FUNCTION fcHMIBit : BOOL
VAR_INPUT
	bInToggle:BOOL;
	bInLatch:BOOL;
END_VAR
VAR_IN_OUT
	bHMI:BOOL;
	bPLC:BOOL;
END_VAR

(*set bPLC when bHMI set*)

IF bHMI AND NOT(bPLC) THEN
	bPLC:=1;
	bHMI:=0;
END_IF

END_FUNCTION

(* stored: Version 1.1.0.1, ProductVersion 3.1.4024.11
   POU fcHMIBit: Id {aca13fec-2890-4eea-aa0d-7e1b55cb41c9}, SpecialFunc None *)
